// TIA Portal V20 export
FUNCTION_BLOCK "Simulation_Interface_STK2"   // FB200, LAD
// stored: Access Published, MemoryReserve 100, SetENOAutomatically false
   VAR_INPUT
      otherSTKDone : Bool;
      resetting : Bool;   // resetting is unit state
      jrDetectUnused : Bool;
      I2S : "LER_typeInspectionToStack";
   END_VAR
   VAR_OUTPUT
      done : Bool;
      S2I : "LER_typeStackToInspection";
   END_VAR
   VAR RETAIN
      simulationData { ExternalAccessible := 'False'; ExternalVisible := 'False'; ExternalWritable := 'False'} : "LER_typeCommonData";   // TCP/IP STK data
   END_VAR
   VAR
      instTON { S7_SetPoint := 'True'} : Array[0..9] of TON_TIME;
      statDone : Bool;
      statBit : Array[0..1] of Bool;
   END_VAR
   VAR CONSTANT
      interfaceDelayTime : Time := T#500ms;
      startDelayTime : Time := T#0s;
   END_VAR
   VAR_TEMP   // added for the SCL form of the ladder/FBD networks
      _w1 : Bool;
   END_VAR
BEGIN

REGION Network 1: Unload request
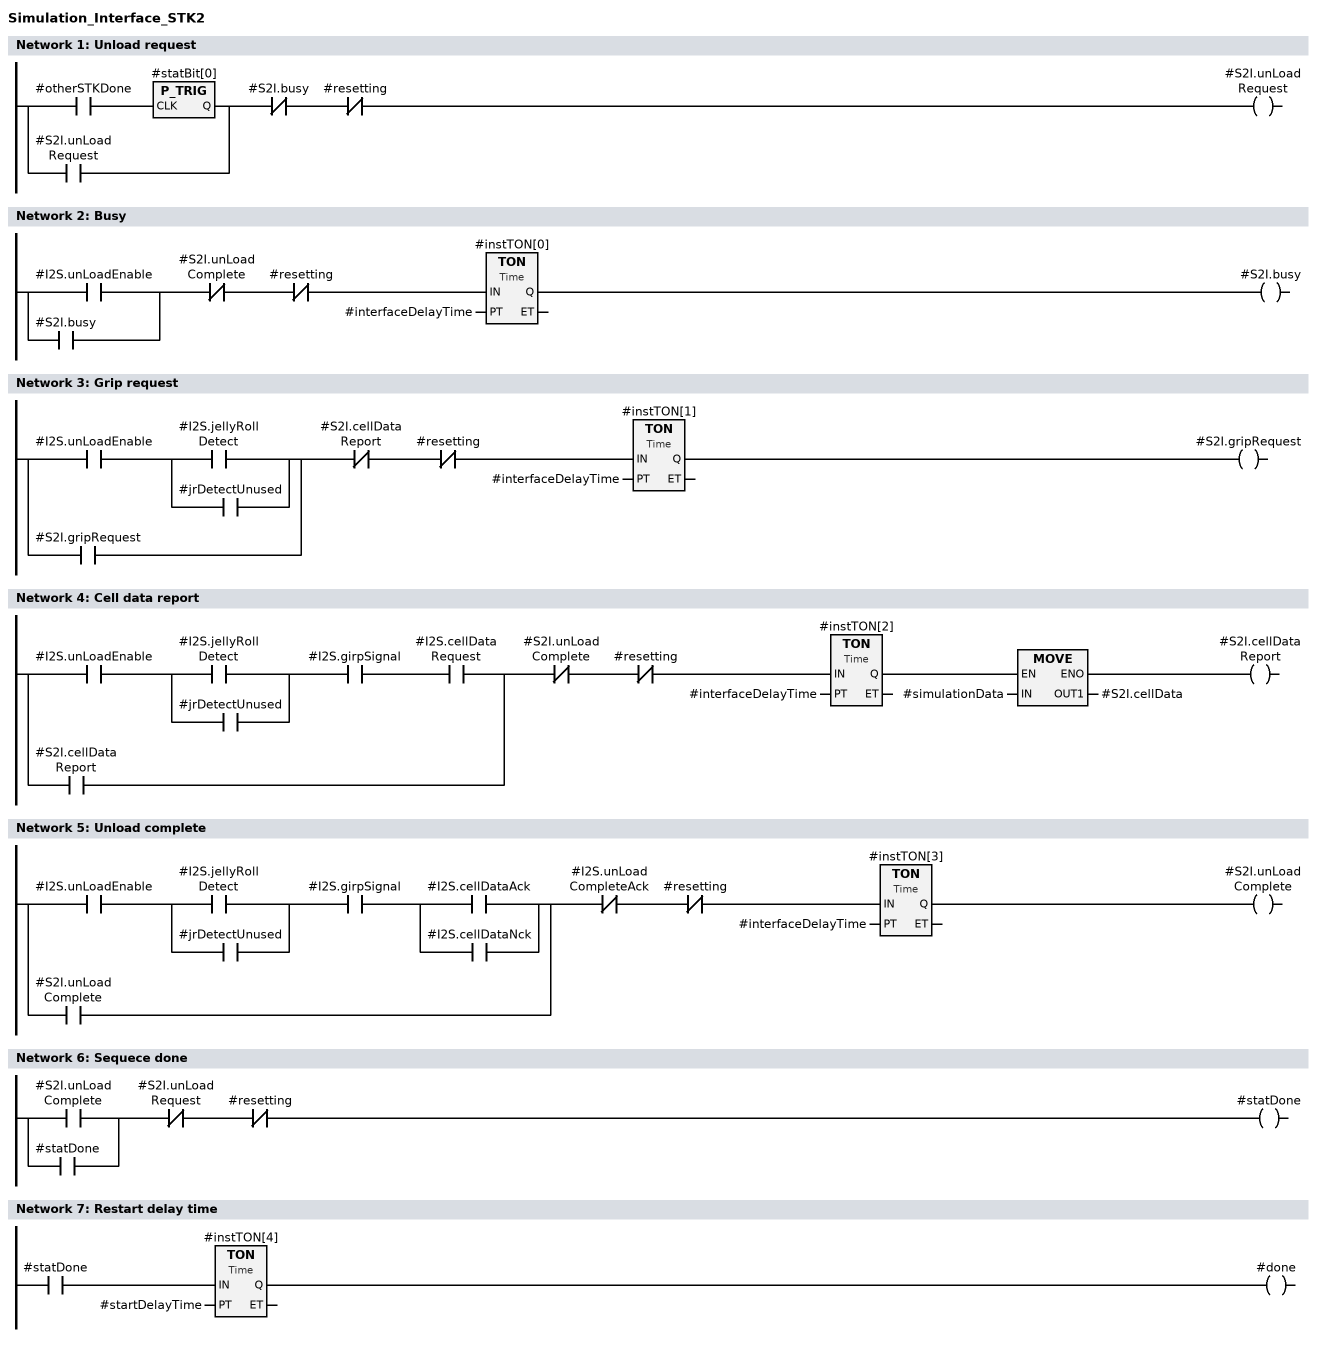
   RUNG wire#powerrail
      Contact( #otherSTKDone )
      P_Trig( #statBit[0] )
      wire#w1
      I_Contact( #S2I.busy )
      I_Contact( #resetting )
      Coil( #S2I.unLoadRequest )
   END_RUNG
   RUNG wire#powerrail
      Contact( #S2I.unLoadRequest )
   END_RUNG wire#w1
   // the same network as SCL:
   #_w1 := #otherSTKDone AND NOT #statBit[0];   // rising edge
   #statBit[0] := #otherSTKDone;
   #S2I.unLoadRequest := (#_w1 OR #S2I.unLoadRequest) AND NOT #S2I.busy AND NOT #resetting;
END_REGION

REGION Network 2: Busy
   RUNG wire#powerrail
      Contact( #I2S.unLoadEnable )
      wire#w1
      I_Contact( #S2I.unLoadComplete )
      I_Contact( #resetting )
      { S7_Templates := "time_type := Time" } #instTON[0].TON(pt := #interfaceDelayTime, et =>)
      Coil( #S2I.busy )
   END_RUNG
   RUNG wire#powerrail
      Contact( #S2I.busy )
   END_RUNG wire#w1
   // the same network as SCL:
   #instTON[0].TON(IN := (#I2S.unLoadEnable OR #S2I.busy) AND NOT #S2I.unLoadComplete AND NOT #resetting,
                   PT := #interfaceDelayTime);
   #S2I.busy := #instTON[0].Q;
END_REGION

REGION Network 3: Grip request
   RUNG wire#powerrail
      Contact( #I2S.unLoadEnable )
      wire#w1
      Contact( #I2S.jellyRollDetect )
      wire#w2
      I_Contact( #S2I.cellDataReport )
      I_Contact( #resetting )
      { S7_Templates := "time_type := Time" } #instTON[1].TON(pt := #interfaceDelayTime, et =>)
      Coil( #S2I.gripRequest )
   END_RUNG
   RUNG wire#w1
      Contact( #jrDetectUnused )
   END_RUNG wire#w2
   RUNG wire#powerrail
      Contact( #S2I.gripRequest )
   END_RUNG wire#w2
   // the same network as SCL:
   #instTON[1].TON(IN := ((#I2S.unLoadEnable AND (#I2S.jellyRollDetect OR #jrDetectUnused)) OR #S2I.gripRequest) AND NOT #S2I.cellDataReport AND NOT #resetting,
                   PT := #interfaceDelayTime);
   #S2I.gripRequest := #instTON[1].Q;
END_REGION

REGION Network 4: Cell data report
   RUNG wire#powerrail
      Contact( #I2S.unLoadEnable )
      wire#w1
      Contact( #I2S.jellyRollDetect )
      wire#w2
      Contact( #I2S.girpSignal )
      Contact( #I2S.cellDataRequest )
      wire#w3
      I_Contact( #S2I.unLoadComplete )
      I_Contact( #resetting )
      { S7_Templates := "time_type := Time" } #instTON[2].TON(pt := #interfaceDelayTime, et =>)
      Move(in := #simulationData, out1 => #S2I.cellData)
      Coil( #S2I.cellDataReport )
   END_RUNG
   RUNG wire#w1
      Contact( #jrDetectUnused )
   END_RUNG wire#w2
   RUNG wire#powerrail
      Contact( #S2I.cellDataReport )
   END_RUNG wire#w3
   // the same network as SCL:
   #instTON[2].TON(IN := ((#I2S.unLoadEnable AND (#I2S.jellyRollDetect OR #jrDetectUnused) AND #I2S.girpSignal AND #I2S.cellDataRequest) OR #S2I.cellDataReport) AND NOT #S2I.unLoadComplete AND NOT #resetting,
                   PT := #interfaceDelayTime);
   IF #instTON[2].Q THEN #S2I.cellData := #simulationData; END_IF;
   #S2I.cellDataReport := #instTON[2].Q;
END_REGION

REGION Network 5: Unload complete
   RUNG wire#powerrail
      Contact( #I2S.unLoadEnable )
      wire#w1
      Contact( #I2S.jellyRollDetect )
      wire#w2
      Contact( #I2S.girpSignal )
      wire#w3
      Contact( #I2S.cellDataAck )
      wire#w4
      I_Contact( #I2S.unLoadCompleteAck )
      I_Contact( #resetting )
      { S7_Templates := "time_type := Time" } #instTON[3].TON(pt := #interfaceDelayTime, et =>)
      Coil( #S2I.unLoadComplete )
   END_RUNG
   RUNG wire#w1
      Contact( #jrDetectUnused )
   END_RUNG wire#w2
   RUNG wire#w3
      Contact( #I2S.cellDataNck )
   END_RUNG wire#w4
   RUNG wire#powerrail
      Contact( #S2I.unLoadComplete )
   END_RUNG wire#w4
   // the same network as SCL:
   #instTON[3].TON(IN := ((#I2S.unLoadEnable AND (#I2S.jellyRollDetect OR #jrDetectUnused) AND #I2S.girpSignal AND (#I2S.cellDataAck OR #I2S.cellDataNck)) OR #S2I.unLoadComplete) AND NOT #I2S.unLoadCompleteAck AND NOT #resetting,
                   PT := #interfaceDelayTime);
   #S2I.unLoadComplete := #instTON[3].Q;
END_REGION

REGION Network 6: Sequece done
   RUNG wire#powerrail
      Contact( #S2I.unLoadComplete )
      wire#w1
      I_Contact( #S2I.unLoadRequest )
      I_Contact( #resetting )
      Coil( #statDone )
   END_RUNG
   RUNG wire#powerrail
      Contact( #statDone )
   END_RUNG wire#w1
   // the same network as SCL:
   #statDone := (#S2I.unLoadComplete OR #statDone) AND NOT #S2I.unLoadRequest AND NOT #resetting;
END_REGION

REGION Network 7: Restart delay time
   RUNG wire#powerrail
      Contact( #statDone )
      { S7_Templates := "time_type := Time" } #instTON[4].TON(pt := #startDelayTime, et =>)
      Coil( #done )
   END_RUNG
   // the same network as SCL:
   #instTON[4].TON(IN := #statDone, PT := #startDelayTime);
   #done := #instTON[4].Q;
END_REGION
END_FUNCTION_BLOCK
